// TwinCAT 3 PLC project Untitled1
// ProgramVersion: 3.1.4023.0
// libraries:
//   Tc2_Standard, * (Beckhoff Automation GmbH)
//   Tc2_System, * (Beckhoff Automation GmbH)
//   Tc3_Module, * (Beckhoff Automation GmbH)
// project tree:
//   DUTs/ BIT8_ARRAY.TcDUT, TaskList.TcDUT
//   / GlobalTextList.TcGTLO, PlcTask.TcTTO
//   POUs/ MAIN.TcPOU, MAIN_obsolete.TcPOU, Robot.TcPOU, RobotLadder.TcPOU
// real-time tasks:
//   TASK PlcTask: cycle T#10ms, priority 20, ADS port 350
//   TASK PlcTask1: cycle T#10ms, priority 21, ADS port 351
// I/O:
//   DEVICE Device 4 (EtherCAT), AmsNetId 192.168.101.188.5.1
//     Box 5 (EP1008-0001) [EP1008-0001 8 Ch. Dig. Input 24V, 3ms, M8]
//   DEVICE Device 1 (EtherCAT), AmsNetId 192.168.101.188.2.1
//     Term 1 (EK1200) [EK1200-5000 EtherCAT Power supply (2A E-Bus)]
//       Term 2 (EL2809) [EL2809 16Ch. Dig. Output 24V, 0.5A]
//       Term 3 (EL6695) [EL6695 EtherCAT Bridge terminal (Primary)]
//       Term 4 (EL9011) [EL9011 End Terminal]
// variable links:
//   Untitled1/Untitled1 Instance <-> Device 1 (EtherCAT)/Term 1 (EK1200)/Term 3 (EL6695)
//     PlcTask Inputs/MAIN.robot1.rangefinderReading <-> IO Inputs/buffer_2
//     PlcTask Inputs/MAIN.robot1.statusReg <-> IO Inputs/buffer
//     PlcTask Outputs/MAIN.robot1.cmd <-> IO Outputs/buffer
//     PlcTask Outputs/MAIN.robot1.moveDist <-> IO Outputs/buffer_6
//   Untitled1/Untitled1 Instance <-> Device 4 (EtherCAT)/Box 5 (EP1008-0001)
//     PlcTask Inputs/MAIN.sensorBlock/bit1 <-> Channel 2/Input

CONFIGURATION Untitled1
    RESOURCE PLC ON TwinCAT3
        TASK PlcTask(INTERVAL := T#10ms, PRIORITY := 20);
        PROGRAM MAIN WITH PlcTask : MAIN;
    END_RESOURCE
END_CONFIGURATION

// ---- DUTs/BIT8_ARRAY.TcDUT
TYPE BIT8_ARRAY :
STRUCT
	bit0 : BIT;
	bit1 : BIT;
	bit2 : BIT;
	bit3 : BIT;
	bit4 : BIT;
	bit5 : BIT;
	bit6 : BIT;
	bit7 : BIT;
END_STRUCT
END_TYPE

// ---- DUTs/TaskList.TcDUT
{attribute 'qualified_only'}
{attribute 'strict'}
TYPE TaskList :
(
	IDLE, 
	HOME:=21,
	POS1, 
	POS2, 
	MOVE_UP, 
	MOVE_DOWN
)WORD;
END_TYPE

// ---- POUs/MAIN.TcPOU
PROGRAM MAIN
VAR
	robot1 : RobotLadder;
	robot2 : Robot;
	sensorBlock AT %I* : BIT8_ARRAY;
	//test : MDP5001_0_A368DC73;
END_VAR

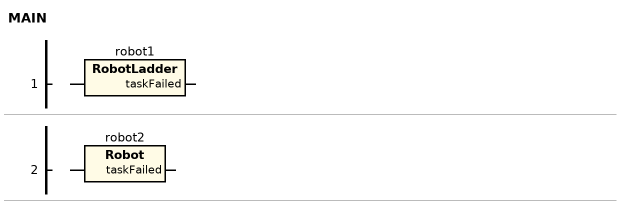
// NETWORK 1
robot1(); // RobotLadder

// NETWORK 2
robot2(); // Robot

END_PROGRAM

// ---- POUs/RobotLadder.TcPOU
FUNCTION_BLOCK RobotLadder
VAR_OUTPUT
	taskFailed : BOOL;
END_VAR
VAR
	cmd AT %Q* : TaskList; //server writes directly to this
	moveDist AT %Q* : WORD;
	
	statusReg AT %I* : UINT;
	
	rangefinderReading AT %I* : UINT;
	
	bAtHome AT %I* : BOOL;
	bAtPos1 AT %I* : BOOL;
	bAtPos2 AT %I* : BOOL;
	bMovedUp AT %I* : BOOL;
	bMovedDown AT %I* : BOOL;
	
	bMoving AT %I* : BOOL;

	timeout : TON;
	step : (IDLE, EXECUTE, FINISHED);
	done : BOOL;
END_VAR
VAR // added by the converter: edge detectors and wires of the graphical bodies
    _w1, _w2, _w3, _w4 : BOOL;
END_VAR

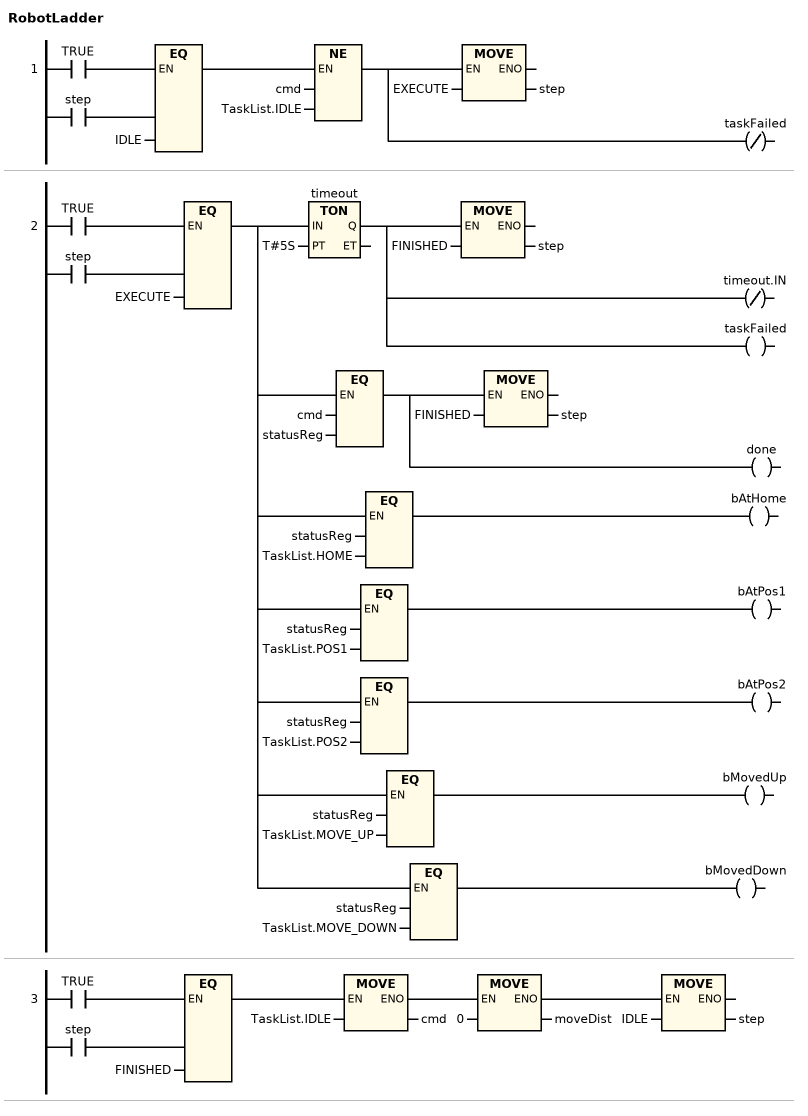
// NETWORK 1
_w1 := step = IDLE AND cmd <> TaskList.IDLE;
IF _w1 THEN step := EXECUTE; END_IF
taskFailed := NOT _w1;

// NETWORK 2
_w2 := step = EXECUTE;
timeout(IN := _w2, PT := T#5S); // TON
IF timeout.Q THEN step := FINISHED; END_IF
timeout.IN := NOT timeout.Q;
taskFailed := timeout.Q;
_w3 := _w2 AND cmd = statusReg;
IF _w3 THEN step := FINISHED; END_IF
done := _w3;
bAtHome := _w2 AND statusReg = TaskList.HOME;
bAtPos1 := _w2 AND statusReg = TaskList.POS1;
bAtPos2 := _w2 AND statusReg = TaskList.POS2;
bMovedUp := _w2 AND statusReg = TaskList.MOVE_UP;
bMovedDown := _w2 AND statusReg = TaskList.MOVE_DOWN;

// NETWORK 3
_w4 := step = FINISHED;
IF _w4 THEN cmd := TaskList.IDLE; END_IF
IF _w4 THEN moveDist := 0; END_IF
IF _w4 THEN step := IDLE; END_IF

END_FUNCTION_BLOCK

// ---- POUs/Robot.TcPOU
FUNCTION_BLOCK Robot
VAR_OUTPUT
	taskFailed : BOOL;
END_VAR
VAR
	cmd AT %Q* : TaskList; //server writes directly to this
	moveDist AT %Q* : WORD;
	
	statusReg AT %I* : UINT;
	
	rangefinderReading AT %I* : BYTE;
	
	bAtHome AT %I* : BOOL;
	bAtPos1 AT %I* : BOOL;
	bAtPos2 AT %I* : BOOL;	
	bMovedUp AT %I* : BOOL;
	bMovedDown AT %I* : BOOL;
	
	bMoving AT %I* : BOOL;
	
	timeout : TON;
	step : (IDLE, EXECUTE, FINISHED);
	done : BOOL;
END_VAR

CASE step OF
	IDLE:
		IF cmd <> TaskList.IDLE THEN
			taskFailed := FALSE;
			step := EXECUTE;
		END_IF
		
	EXECUTE: //perform task
		timeout(IN:= , PT:= T#5S, Q=> , ET=> );
		timeout.IN := TRUE;
		
		IF timeout.Q THEN
			timeout.IN := FALSE;
			taskFailed := TRUE;
			step := FINISHED;
			RETURN;
		END_IF
		
		bAtHome := statusReg = TaskList.HOME;
		bAtPos1 := statusReg = TaskList.POS1;
		bAtPos2 := statusReg = TaskList.POS2;
		bMovedUp := statusReg = TaskList.MOVE_UP;
		bMovedDown := statusReg = TaskList.MOVE_DOWN;
		
		done := statusReg = cmd;

		IF done THEN
			timeout.IN := FALSE;
			step := FINISHED;
		END_IF
	
	FINISHED: //task done, reset
		cmd := 0;
		moveDist := 0;
		step := IDLE;
END_CASE

END_FUNCTION_BLOCK

// ---- POUs/MAIN_obsolete.TcPOU
PROGRAM MAIN_obsolete
VAR
	robot1 : RobotLadder;
	robot2 : Robot;
	sensorBlock AT %I* : BIT8_ARRAY;
	//test : MDP5001_0_A368DC73;
END_VAR

robot1();
robot2();

END_PROGRAM
